ABB RobotStudio station: proyecto.rsstnx

Station Project1 (saved by RobotStudio 25.5.11605.0)
Controller IRB140_6_81
  mechanical unit ROB_1: IRB140_6_81_C_03, 6 joints, base frame (0, 0, 0) mm
Layout (positions relative to the parent item):
  - IRB140_6_81_C_03 [mechanism, from %ABB.RobotStudio.Models.IRB140%\IRB140_6_81_C_G_03.rslib] at (0, 0, 0) mm; joint values [0, 0.6343, -0.3791, 0, 0.7304, 0] (rad or m)
Targets, tools, work objects and paths stored in the station, written as RAPID:
! task T_ROB1
MODULE Module1
  CONST robtarget Target_30:=[[506.291651246,0,679.5],[0.5,0,0.866025404,0],[0,0,0,0],[9E+09,9E+09,9E+09,9E+09,9E+09,9E+09]];
  PROC Path_10()
    MoveJ Target_30,v500,fine,tool0\WObj:=wobj0;
    MoveJ Target_10_2,v500,fine,tool0\WObj:=wobj0;
    MoveL Target_10_4,vmax,fine,tool0\WObj:=wobj0;
    MoveJ Target_30,v500,z0,tool0\WObj:=wobj0;
  ENDPROC
ENDMODULE

